FUNCTION_BLOCK FB_Module

VAR_INPUT
	dr		: REFERENCE TO FB_Director;
	ID		: BYTE; 		// identificador de la unidad funcional (el módulo)
	Name	: STRING;		// Nombre del módulo (para erroers)
	Descr	: STRING; 		// Descripción del módulo (para tooltips)
	
	IC: BOOL;
	Execute: BOOL;
	Ack: BOOL;

END_VAR
VAR_OUTPUT
	Ready: BOOL;
	Failure: BOOL;
	Done: BOOL;
	IsActive: BOOL;
END_VAR

// TODO AÑADIR UN METODO GEMMA QUE SE INVOQUE DESDE PROCESSCYCLE PARA TRATAMIENTO DE PARADA, PAUSA...
VAR_INPUT
END_VAR

VAR_OUTPUT
	//ctOut: S_ControllerOutput;
//	IC: BOOL;
//	Done: BOOL;
END_VAR

METHOD InitialConditions : BOOL
VAR_INPUT
END_VAR
InitialConditions := TRUE;
END_METHOD

METHOD ProcessCycle : BOOL 
VAR_INPUT
	dr	: REFERENCE TO FB_Director;
END_VAR
IsActive := FALSE;
END_METHOD

END_FUNCTION_BLOCK

(* stored: Version 1.1.0.1, ProductVersion 3.1.4024.6
   POU FB_Module: Id {cba3fcf8-6c8d-4174-8dda-f766b8b369f3}, SpecialFunc None
   Method InitialConditions: Id {569290b0-7483-4183-aad6-de676bf056ec}
   Method ProcessCycle: Id {9383c466-5ef4-45f2-bc56-c203e01f0aa7} *)
